FUNCTION_BLOCK TEST
VAR_INPUT
END_VAR
VAR_OUTPUT
END_VAR
VAR
END_VAR

END_FUNCTION_BLOCK

(* stored: Version 1.1.0.1, ProductVersion 3.1.4024.14
   POU TEST: Id {738b160f-042e-4038-adcd-a65b7bb2eca0}, SpecialFunc None *)
